// TIA Portal V19 export
FUNCTION_BLOCK "IFM_AL2221_PD"   // FB119, STL
TITLE = IFM AL2221 IO-Link VendorID 310, DeviceID 1314, Process Data
{ S7_Optimized_Access := 'TRUE' }
AUTHOR : AFL
FAMILY : IO_Link
NAME : AL2221
// IO_Config Byte 
//  ****************
//  Bit 0 to 7 represents the IO configuration of Ports
//  X1.0 to X1.7, where Input ports are False and 
//  output ports are True.
//  That is, B#16#01 means only Port 1.0 is an Output
//  port and the rest are Input ports.
// 
//  Device status
//  *************
//  0 Everything is OK
//  1  Maintenance required
//  2 Out of specification
//  3 Functional check
//  4 Failure
// stored: AutoNumber false, MemoryReserve 100
   VAR_INPUT
      Addr : Int;   // First Byte address of 4 byte address space
      IO_Config : Byte;   // See block comments
      DO_X1_0_p4 : Bool;   // Digit Ouput X1.0 - pin 4
      DO_X1_0_p2 : Bool;   // Digit Ouput X1.0 - pin 2
      DO_X1_1_p4 : Bool;   // Digit Ouput X1.1 - pin 4
      DO_X1_1_p2 : Bool;   // Digit Ouput X1.1 - pin 2
      DO_X1_2_p4 : Bool;   // Digit Ouput X1.2 - pin 4
      DO_X1_2_p2 : Bool;   // Digit Ouput X1.2 - pin 2
      DO_X1_3_p4 : Bool;   // Digit Ouput X1.3 - pin 4
      DO_X1_3_p2 : Bool;   // Digit Ouput X1.3 - pin 2
      DO_X1_4_p4 : Bool;   // Digit Ouput X1.4 - pin 4
      DO_X1_4_p2 : Bool;   // Digit Ouput X1.4 - pin 2
      DO_X1_5_p4 : Bool;   // Digit Ouput X1.5 - pin 4
      DO_X1_5_p2 : Bool;   // Digit Ouput X1.5 - pin 2
      DO_X1_6_p4 : Bool;   // Digit Ouput X1.6 - pin 4
      DO_X1_6_p2 : Bool;   // Digit Ouput X1.6 - pin 6
      DO_X1_7_p4 : Bool;   // Digit Ouput X1.7 - pin 4
      DO_X1_7_p2 : Bool;   // Digit Ouput X1.7 - pin 7
   END_VAR
   VAR_OUTPUT
      DI_X1_0_p4 : Bool;   // Digit Input X1.0 - pin 4
      DI_X1_0_p2 : Bool;   // Digit Input X1.0 - pin 2
      DI_X1_1_p4 : Bool;   // Digit Input X1.1 - pin 4
      DI_X1_1_p2 : Bool;   // Digit Input X1.1 - pin 2
      DI_X1_2_p4 : Bool;   // Digit Input X1.2 - pin 4
      DI_X1_2_p2 : Bool;   // Digit Input X1.2 - pin 2
      DI_X1_3_p4 : Bool;   // Digit Input X1.3 - pin 4
      DI_X1_3_p2 : Bool;   // Digit Input X1.3 - pin 2
      DI_X1_4_p4 : Bool;   // Digit Input X1.4 - pin 4
      DI_X1_4_p2 : Bool;   // Digit Input X1.4 - pin 2
      DI_X1_5_p4 : Bool;   // Digit Input X1.5 - pin 4
      DI_X1_5_p2 : Bool;   // Digit Input X1.5 - pin 2
      DI_X1_6_p4 : Bool;   // Digit Input X1.6 - pin 4
      DI_X1_6_p2 : Bool;   // Digit Input X1.6 - pin 6
      DI_X1_7_p4 : Bool;   // Digit Input X1.7 - pin 4
      DI_X1_7_p2 : Bool;   // Digit Input X1.7 - pin
      SC_X1_0 : Bool;   // Short Circuit on X1.0
      SC_X1_1 : Bool;   // Short Circuit on X1.1
      SC_X1_2 : Bool;   // Short Circuit on X1.2
      SC_X1_3 : Bool;   // Short Circuit on X1.3
      SC_X1_4 : Bool;   // Short Circuit on X1.4
      SC_X1_5 : Bool;   // Short Circuit on X1.5
      SC_X1_6 : Bool;   // Short Circuit on X1.6
      SC_X1_7 : Bool;   // Short Circuit on X1.7
      UV_UA : Bool;   // Undervoltage of UA power supply
      UV_UAi : Bool;   // Undervoltage of UAi power supply
      SC_Pin1 : Bool;   // Short Circuit on sensor power supply
      DeviceStatus : Byte;   // See Block Comment
      EquipID : Byte;   // See Block Comment
      O_DI4 : Bool;   // Output signal status Pin 4
      O_DI2 : Bool;   // Output signal status Pin 2
      O_DA : Bool;   // Output device recognised
      O_DE : Bool;   // Output device error event has appeared
      O_PQ : Bool;   // Output port qualifer proces data valid
   END_VAR
   VAR_TEMP
      tmp_IO_Config : Byte;   // Local Byte 0
      tmp_spare : Byte;   // Local Byte 1
      tmp_InputWord : Word;   // LB2 = p4's LB3 = p2's
      tmp_sc : Word;   // LB4 = sc , LB5 = UA
      TW_Flag : Word;
   END_VAR
BEGIN

NETWORK
TITLE = 
// Get first byte address
      L     #Addr;
      SLW   3;
      LAR1;

// IO Config Byte
      L     #IO_Config;
      T     #tmp_IO_Config;

// ************** AL2221 Outputs / Function Intputs*******************

// DO X1.0
      A     #tmp_IO_Config.%X0;  // IO Config
      A     #DO_X1_0_p4;
      =     Q [AR1, P#2.0];
      A     #tmp_IO_Config.%X0;  // IO Config
      A     #DO_X1_0_p2;
      =     Q [AR1, P#3.0];
// DO X1.1
      A     #tmp_IO_Config.%X1;  // IO Config
      A     #DO_X1_1_p4;
      =     Q [AR1, P#2.1];
      A     #tmp_IO_Config.%X1;  // IO Config
      A     #DO_X1_1_p2;
      =     Q [AR1, P#3.1];
// DO X1.2
      A     #tmp_IO_Config.%X2;  // IO Config
      A     #DO_X1_2_p4;
      =     Q [AR1, P#2.2];
      A     #tmp_IO_Config.%X2;  // IO Config
      A     #DO_X1_2_p2;
      =     Q [AR1, P#3.2];
// DO X1.3
      A     #tmp_IO_Config.%X3;  // IO Config
      A     #DO_X1_3_p4;
      =     Q [AR1, P#2.3];
      A     #tmp_IO_Config.%X3;  // IO Config
      A     #DO_X1_3_p2;
      =     Q [AR1, P#3.3];
// DO X1.4
      A     #tmp_IO_Config.%X4;  // IO Config
      A     #DO_X1_4_p4;
      =     Q [AR1, P#2.4];
      A     #tmp_IO_Config.%X4;  // IO Config
      A     #DO_X1_4_p2;
      =     Q [AR1, P#3.4];
// DO X1.5;
      A     #tmp_IO_Config.%X5;  // IO Config
      A     #DO_X1_5_p4;
      =     Q [AR1, P#2.5];
      A     #tmp_IO_Config.%X5;  // IO Config
      A     #DO_X1_5_p2;
      =     Q [AR1, P#3.5];
// DO X1.6
      A     #tmp_IO_Config.%X6;  // IO Config
      A     #DO_X1_6_p4;
      =     Q [AR1, P#2.6];
      A     #tmp_IO_Config.%X6;  // IO Config
      A     #DO_X1_6_p2;
      =     Q [AR1, P#3.6];
// DO X1.7
      A     #tmp_IO_Config.%X7;  // IO Config
      A     #DO_X1_7_p4;
      =     Q [AR1, P#2.7];
      A     #tmp_IO_Config.%X7;  // IO Config
      A     #DO_X1_7_p2;
      =     Q [AR1, P#3.7];
// *** Write Output Image to periferal Output image

      L     QW [AR1, P#2.0];
      T     QW [AR1, P#2.0];


// ************** AL2221 Inputs / Function Outputs*******************

// Device Status
      L     IB [AR1, P#0.0];
      T     #DeviceStatus;

// Equipment Specific ID
      L     IB [AR1, P#1.0];
      T     #EquipID;

// Get Input word
      L     IW [AR1, P#2.0];
      T     #tmp_InputWord;

// DI X1.0
      AN    #tmp_IO_Config.%X0;  // IO Config
      A     #tmp_InputWord.%X0;
      =     #DI_X1_0_p2;
      AN    #tmp_IO_Config.%X0;  // IO Config
      A     #tmp_InputWord.%X8;
      =     #DI_X1_0_p4;

// DI X1.1
      AN    #tmp_IO_Config.%X1;  // IO Config
      A     #tmp_InputWord.%X1;
      =     #DI_X1_1_p2;
      AN    #tmp_IO_Config.%X1;  // IO Config
      A     #tmp_InputWord.%X9;
      =     #DI_X1_1_p4;

// DI X1.2
      AN    #tmp_IO_Config.%X2;  // IO Config
      A     #tmp_InputWord.%X2;
      =     #DI_X1_2_p2;
      AN    #tmp_IO_Config.%X2;  // IO Config
      A     #tmp_InputWord.%X10;
      =     #DI_X1_2_p4;

// DI X1.3
      AN    #tmp_IO_Config.%X3;  // IO Config
      A     #tmp_InputWord.%X3;
      =     #DI_X1_3_p2;
      AN    #tmp_IO_Config.%X3;  // IO Config
      A     #tmp_InputWord.%X11;
      =     #DI_X1_3_p4;

// DI X1.4
      AN    #tmp_IO_Config.%X4;  // IO Config
      A     #tmp_InputWord.%X4;
      =     #DI_X1_4_p2;
      AN    #tmp_IO_Config.%X4;  // IO Config
      A     #tmp_InputWord.%X12;
      =     #DI_X1_4_p4;

// DI X1.5
      AN    #tmp_IO_Config.%X5;  // IO Config
      A     #tmp_InputWord.%X5;
      =     #DI_X1_5_p2;
      AN    #tmp_IO_Config.%X5;  // IO Config
      A     #tmp_InputWord.%X13;
      =     #DI_X1_5_p4;

// DI X1.6
      AN    #tmp_IO_Config.%X6;  // IO Config
      A     #tmp_InputWord.%X6;
      =     #DI_X1_6_p2;
      AN    #tmp_IO_Config.%X6;  // IO Config
      A     #tmp_InputWord.%X14;
      =     #DI_X1_6_p4;

// DI X1.7
      AN    #tmp_IO_Config.%X7;  // IO Config
      A     #tmp_InputWord.%X7;
      =     #DI_X1_7_p2;
      AN    #tmp_IO_Config.%X7;  // IO Config
      A     #tmp_InputWord.%X15;
      =     #DI_X1_7_p4;

// Get Short Circuit Status Input word
      L     IW [AR1, P#4.0];
      T     #tmp_sc;
// SC X1.0
      A     #tmp_sc.%X8;
      =     #SC_X1_0;
// SC X1.1
      A     #tmp_sc.%X9;
      =     #SC_X1_1;
// SC X1.2
      A     #tmp_sc.%X10;
      =     #SC_X1_2;
// SC X1.3
      A     #tmp_sc.%X11;
      =     #SC_X1_3;
// SC X1.4
      A     #tmp_sc.%X12;
      =     #SC_X1_4;
// SC X1.5
      A     #tmp_sc.%X13;
      =     #SC_X1_5;
// SC X1.6
      A     #tmp_sc.%X14;
      =     #SC_X1_6;
// SC X1.7
      A     #tmp_sc.%X15;
      =     #SC_X1_7;
// UV_UA;
      A     #tmp_sc.%X7;
      =     #UV_UA;
// UV_UAi
      A     #tmp_sc.%X6;
      =     #UV_UAi;
// SC_Pin1
      A     #tmp_sc.%X5;
      =     #SC_Pin1;

// PQI

      L     IB [AR1, P#6.0];
      T     #TW_Flag;

      L     #TW_Flag;
      L     1;
      AW;
      L     1;
      ==I;
      =     #O_DI4;



      L     #TW_Flag;
      L     2;
      AW;
      L     2;
      ==I;
      =     #O_DI2;

      L     #TW_Flag;
      L     32;
      AW;
      L     32;
      ==I;
      =     #O_DA;

      L     #TW_Flag;
      L     64;
      AW;
      L     64;
      ==I;
      =     #O_DE;


      L     #TW_Flag;
      L     128;
      AW;
      L     128;
      ==I;
      =     #O_PQ;


END_FUNCTION_BLOCK
